# EPICS autosave request: App/Db/qimaging_settings.req
$(P)$(R)qReadoutSpeed
$(P)$(R)qOffset
$(P)$(R)qImageFormat
$(P)$(R)qCoolerActive
